PROGRAM MAIN
VAR
	//Stati
	IN_FUNZIONE: BOOL;
	IN_SMISTAMENTO: BOOL;
	IN_TIMBRATURA: BOOL;
	IN_FORATURA: BOOL;
	PEZZO_BIANCO: BOOL;
	PEZZO_NERO: BOOL;
	
	//Timer
	TON_BIANCO: TON;
	TON_NERO: TON;
	TON_TIMBRATURA: TON;
	TON_FORATURA_1: TON; // Il trapano scende in 2 secondi
	TON_FORATURA_2: TON; // Il trapano risale in 2 secondi

	//Counter
	CTU_BIANCHI: CTU;
	CTU_NERI: CTU;
END_VAR

GestionePulsantiSegnalazioni();
GestioneMotori();
GestioneSmistamento();
GestioneTimbratura();
GestioneForatura();
GestioneConteggio();

ACTION GestioneConteggio:
// NETWORK 1
END_ACTION

ACTION GestioneForatura:
// NETWORK 1
END_ACTION

ACTION GestioneMotori:
// NETWORK 1
END_ACTION

ACTION GestionePulsantiSegnalazioni:
// NETWORK 1
END_ACTION

ACTION GestioneSmistamento:
// NETWORK 1
END_ACTION

ACTION GestioneTimbratura:
// NETWORK 1
END_ACTION

END_PROGRAM

(* stored: Version 1.1.0.1, ProductVersion 3.1.4024.12
   POU MAIN: Id {77ce3c58-9155-42f5-9eb6-c02febfddbf9}, SpecialFunc None
   Action GestioneConteggio: Id {619b20d3-e452-44f5-b626-dfa96b8409ac}
   Action GestioneForatura: Id {231e95f2-6121-4dbc-89e6-afb7e53183f4}
   Action GestioneMotori: Id {9e464890-6681-41a5-8f39-3082d5bac0ef}
   Action GestionePulsantiSegnalazioni: Id {3f00a759-f8d0-455e-af78-03f29b3994ec}
   Action GestioneSmistamento: Id {6f07de2f-68ba-41e8-a08f-d2eacd4f38eb}
   Action GestioneTimbratura: Id {12208fa5-515e-473c-96cd-01596b797502} *)
